FUNCTION_BLOCK TcoLoggerTest EXTENDS TcoCore.TcoObject

END_FUNCTION_BLOCK

(* stored: Version 1.1.0.1
   POU TcoLoggerTest: Id {8aa4f067-688a-0cea-3c82-efe104e2c1f0}, SpecialFunc None *)
